% RSLogix 500 project Digital Rotameter.RSS, saved by version 8.30.00.16 %
PROJECT "UNTITLED"    % processor: Bul.1763 MicroLogix 1100 Series B %

PROGRAM FILES
  LAD 2 "MAIN"  3 rungs
  LAD 3 "SIMULATION"  2 rungs
  LAD 4 "LOGIC"  3 rungs

DATA FILES
  O0 OUTPUT  4 elements
  I1 INPUT  6 elements
  S2 STATUS  66 elements
  B3 BINARY  1 elements
  T4 TIMER  4 elements
  C5 COUNTER  1 elements
  R6 CONTROL  1 elements
  N7 INTEGER  1 elements
  F8 FLOAT  4 elements

LADDER 2 "MAIN"
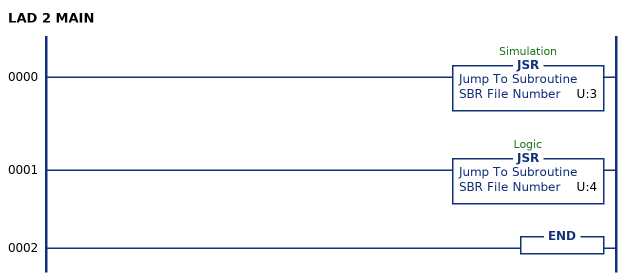
% Rung: 0 %
SOR JSR U:3 EOR
%   U:3  "Simulation" %
% Rung: 1 %
SOR JSR U:4 EOR
%   U:4  "Logic" %
% Rung: 2 %
SOR END EOR

LADDER 3 "SIMULATION"
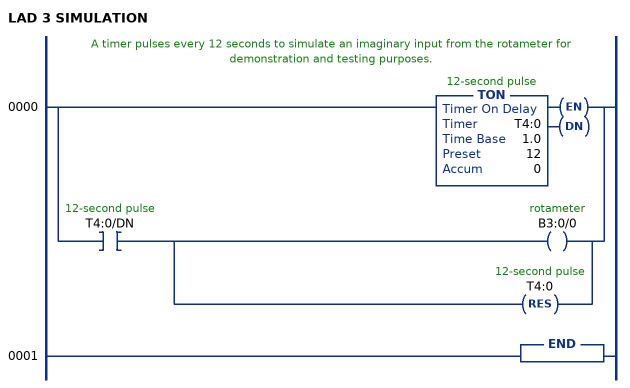
% Rung: 0 %
% A timer pulses every 12 seconds to simulate an imaginary input from the rotameter for demonstration and testing purposes. %
SOR BST TON T4:0 1.0 12 0 NXB XIC T4:0/DN BST OTE B3:0/0 NXB RES T4:0 BND BND EOR
%   T4:0  "12-second pulse" %
%   B3:0/0  "rotameter" %
% Rung: 1 %
SOR END EOR

LADDER 4 "LOGIC"
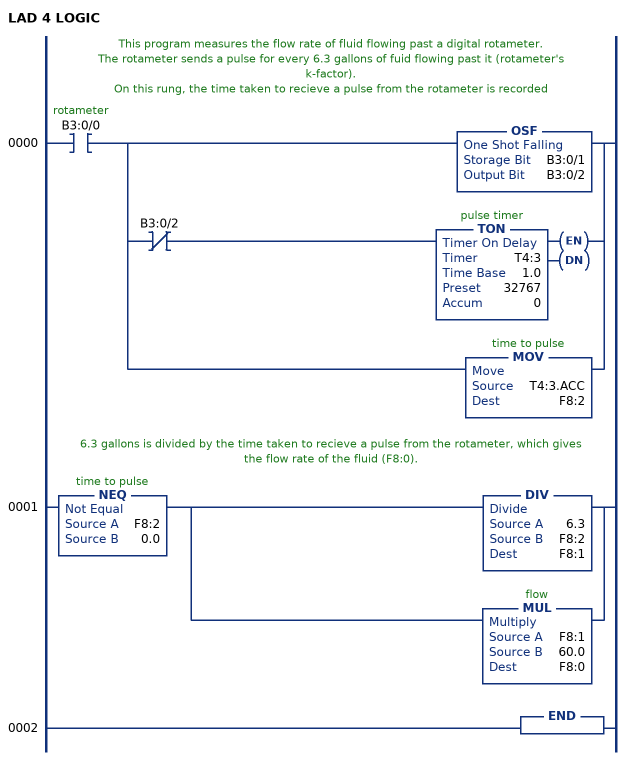
% Rung: 0 %
% This program measures the flow rate of fluid flowing past a digital rotameter.
% The rotameter sends a pulse for every 6.3 gallons of fuid flowing past it (rotameter's k-factor).
% On this rung, the time taken to recieve a pulse from the rotameter is recorded %
SOR XIC B3:0/0 BST OSF B3:0/1 B3:0/2 NXB XIO B3:0/2 TON T4:3 1.0 32767 0 NXB MOV T4:3.ACC F8:2 BND EOR
%   B3:0/0  "rotameter" %
%   T4:3  "pulse timer" %
%   F8:2  "time to pulse" %
% Rung: 1 %
% 6.3 gallons is divided by the time taken to recieve a pulse from the rotameter, which gives the flow rate of the fluid (F8:0). %
SOR NEQ F8:2 0.0 BST DIV 6.3 F8:2 F8:1 NXB MUL F8:1 60.0 F8:0 BND EOR
%   F8:2  "time to pulse" %
%   F8:0  "flow" %
% Rung: 2 %
SOR END EOR

OTHER DOCUMENTED ADDRESSES
  B3:0/4  "ON"
  T4:1  "1-minute timer"

DATA TABLE (non-zero values as saved)
DATA T4
% .PRE .ACC %
% T4:0 % 12 0
% T4:1 % 60 0
% T4:3 % 32767 0
